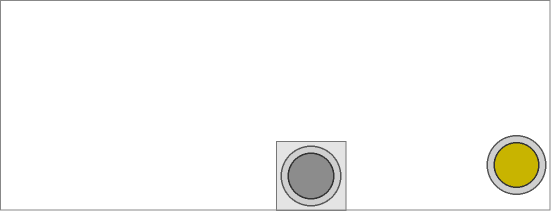
VISUALIZATION Visualization  // 551x211
    PushSwitch (276,141 70x70), variable: GVL.StartButton, behaviour: TOGGLE, style: Switch-PushSwitch-Gray
    Lamp1 (482,130 69x70), variable: GVL.Clamping, style: Lamp-Lamp1-Yellow
END_VISUALIZATION

(* stored: Version 1.1.0.1, ProductVersion 3.1.4024.12
   Visu Visualization: Id {1b60d73f-a5f1-4fba-9c87-21801d9cc17c} *)
